PROGRAM MAIN
VAR
	// print out 'Hello world'
	fbStringBuilder : FB_StringBuilder;
	sResult : STRING;
	bTest : BOOL;
END_VAR

IF bTest THEN
	sResult := fbStringBuilder.Clear()
								.Append('H')
								.Append('e')
								.Append('l')
								.Append('l')
								.Append('o')
								.Append(' ')
								.Append('W')
								.Append('o')
								.Append('r')
								.Append('l')
								.Append('d')
								.ToString();
	bTest := FALSE;
END_IF

END_PROGRAM

(* stored: Version 1.1.0.1, ProductVersion 3.1.4024.12
   POU MAIN: Id {f312f0fa-099f-4c2b-984a-6c47d5371a94}, SpecialFunc None *)
